ORGANIZATION_BLOCK MAIN:OB1
TITLE=PROGRAM COMMENTS
BEGIN
Network 1
LD     SM0.5
=      Q0.0
=      Q0.1
=      Q0.2
=      Q0.3
=      Q0.4
=      Q0.5
=      Q0.6
Network 2
END_ORGANIZATION_BLOCK
INTERRUPT_BLOCK INT_0:INT0
TITLE=INTERRUPT ROUTINE COMMENTS
BEGIN
Network 1 // Network Title
// Network Comment
END_INTERRUPT_BLOCK
